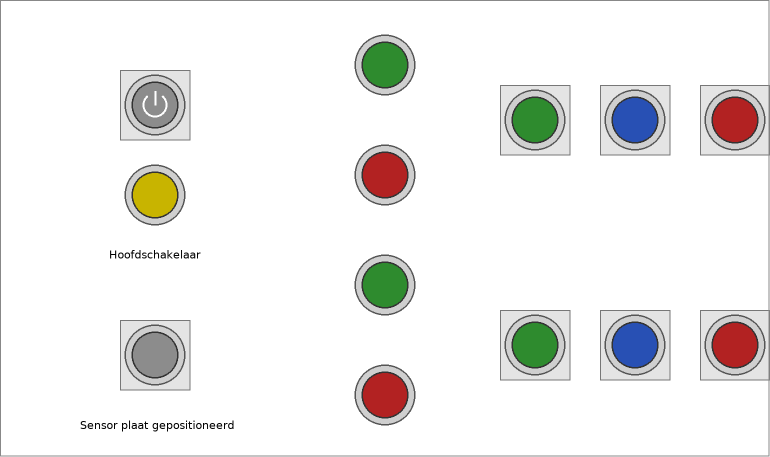
VISUALIZATION Visualization  // 770x457
    Lamp1 (350,30 70x70), variable: GVL.Boor_Start, style: Lamp-Lamp1-Green
    PowerSwitch (120,70 70x70), variable: GVL.Hoofdschakelaar, behaviour: TOGGLE, style: Switch-PowerSwitch-Gray
    Lamp1 (350,140 70x70), variable: GVL.Boor_Retour, style: Lamp-Lamp1-Red
    Lamp1 (350,250 70x70), variable: GVL.Tappen_Start, style: Lamp-Lamp1-Green
    PushSwitchLed (120,320 70x70), variable: GVL.Plaat_Gepositioneerd, behaviour: TOGGLE, style: Switch-PushSwitchLed-Gray
    Lamp1 (120,160 70x70), variable: GVL.Lamp_Hoofdschakelaar, style: Lamp-Lamp1-Yellow
    Label (80,240 150x30), "Hoofdschakelaar"
    Label (66,394 183x63), "Sensor plaat gepositioneerd"
    Lamp1 (350,360 70x70), variable: GVL.Tappen_Retour, style: Lamp-Lamp1-Red
    PushSwitch (500,85 70x70), variable: GVL.Boor_aan, behaviour: TAP, style: Switch-PushSwitch-Green
    PushSwitch (600,85 70x70), variable: GVL.boor_Pos_Bereikt, behaviour: TAP, style: Switch-PushSwitch-Blue
    PushSwitch (700,85 70x70), variable: GVL.boor_uit, behaviour: TAP, style: Switch-PushSwitch-Red
    PushSwitch (500,310 70x70), variable: GVL.Tappen_aan, behaviour: TAP, style: Switch-PushSwitch-Green
    PushSwitch (600,310 70x70), variable: GVL.Tappen_Pos_Bereikt, behaviour: TAP, style: Switch-PushSwitch-Blue
    PushSwitch (700,310 70x70), variable: GVL.Tappen_uit, behaviour: TAP, style: Switch-PushSwitch-Red
END_VISUALIZATION

(* stored: Version 1.1.0.1, ProductVersion 3.1.4024.12
   Visu Visualization: Id {818707b7-945b-4749-9b04-1124db28edfd} *)
